FUNCTION_BLOCK FB_SV
VAR_IN_OUT

END_VAR
VAR_INPUT
	Freigabe_auto			: BOOL;
	Freigabe_Deakt_auto		: BOOL;
	Stellung_Anford_auto	: BOOL;
	Quittierung				: BOOL;
	Parameter_init			: ST_SV_Parameter;
END_VAR
VAR_OUTPUT
	{attribute 'OPC.UA.DA' := '1'}Parameter				: ST_SV_Parameter;			
	{attribute 'OPC.UA.DA' := '1'}Steuerung				: ST_SV_Steuerung;			
	{attribute 'OPC.UA.DA' := '1'}Stellwert				: ST_SV_Stellwert;			
	{attribute 'OPC.UA.DA' := '1'}Zustand					: ST_SV_Zustand;		

END_VAR
VAR
	Zustandscheck			: FB_SV_Zustandscheck;
	Logik					: FB_SV_Logik;
	Ablaufsteuerung			: FB_SV_Ablaufsteuerung;
	QuitTrig				: FB_SetResetFallTrigger;

	SchreibeDaten			: FB_SV_Output;
	OUT_Stellung			AT %Q* : BOOL;
END_VAR

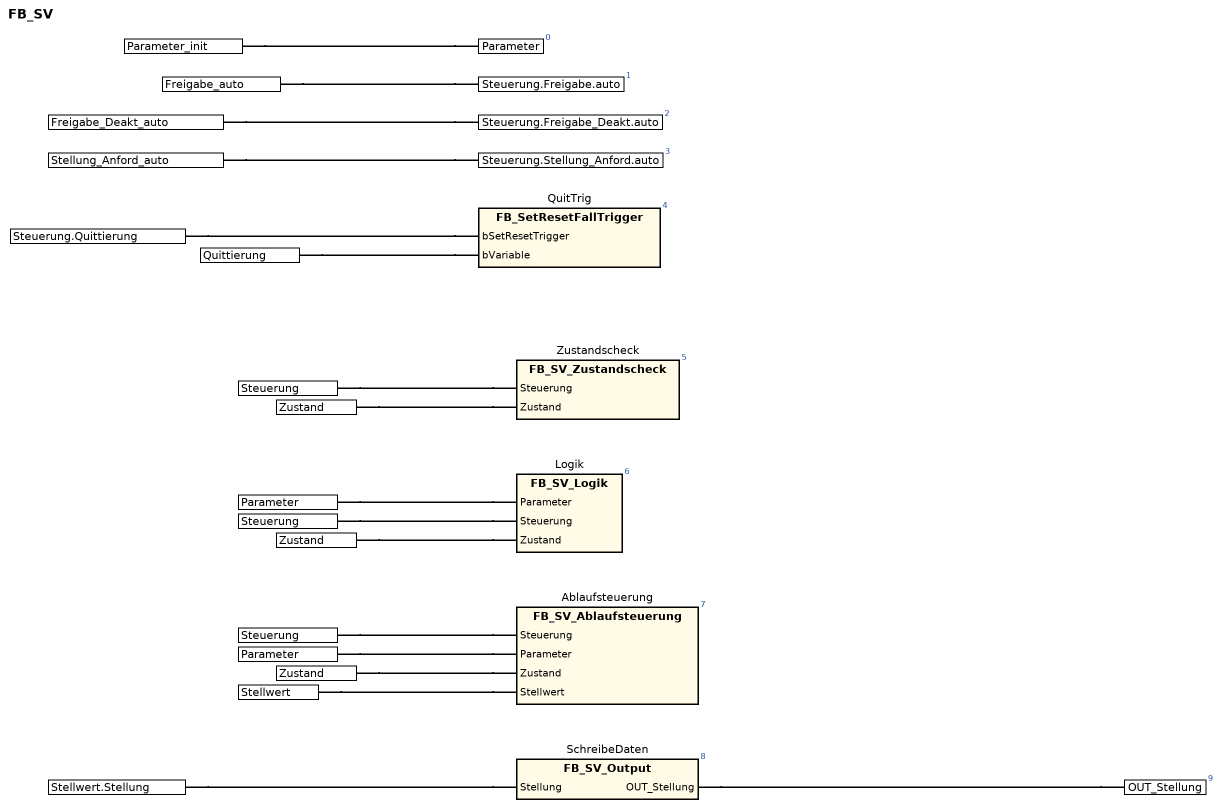
Parameter := Parameter_init;
Steuerung.Freigabe.auto := Freigabe_auto;
Steuerung.Freigabe_Deakt.auto := Freigabe_Deakt_auto;
Steuerung.Stellung_Anford.auto := Stellung_Anford_auto;
QuitTrig(bSetResetTrigger := Steuerung.Quittierung, bVariable := Quittierung); // FB_SetResetFallTrigger
Zustandscheck(Steuerung := Steuerung, Zustand := Zustand); // FB_SV_Zustandscheck
Logik(Parameter := Parameter, Steuerung := Steuerung, Zustand := Zustand); // FB_SV_Logik
Ablaufsteuerung(Steuerung := Steuerung, Parameter := Parameter, Zustand := Zustand, Stellwert := Stellwert); // FB_SV_Ablaufsteuerung
SchreibeDaten(Stellung := Stellwert.Stellung); // FB_SV_Output
OUT_Stellung := SchreibeDaten.OUT_Stellung;

END_FUNCTION_BLOCK

(* stored: Version 1.1.0.1, ProductVersion 3.1.4024.9
   POU FB_SV: Id {8bad8c17-316c-4e05-a9d6-f8f2a3331189}, SpecialFunc None *)
